// TIA Portal V20 export
DATA_BLOCK "DataFromStandard"   // DB128
// stored: Access Published, InstanceOfName Safety.typeDataToSafety, InstanceOfType UDT, Namespace Safety
"Safety.typeDataToSafety"
   // VAR
   //    ackSafetyFromHmi : Int;
   //    ackSafetyGlobal : Bool;
   //    ackFromUnit1 : Bool;
   //    ackSafetyFromMobileHMI : Bool;
   //    resetSafetyFromMobileHMI : Bool;
   //    connectionBoxID_1 : Int;
   //    connectionBoxID_2 : Int;
   //    MobilePanelConnected : Bool;
   //    MobilePannelPermissions : Bool;
   //    "PhmiNo1.Connected" : Bool;
   //    "PhmiNo2.Connected" : Bool;
   //    KeyBoxStatus : Int;
   //    DeselectBA30 : Bool;
   //    DeselectBA40 : Bool;
   //    DeselectBA15 : Bool;
   //    DeselectBA60 : Bool;
   //    PowerOnCommand : Bool;
   //    leftUnwinderRadius : Int;
   //    rightUnwinderRadius : Int;
   //    PhmiCommunicationOK : Bool;
   //    allBrakeTesting : "Safety.typeBrakeTest";
   //    Unwinder_Left_DiaData : "Safety.typeSafetyDia";
   //    Unwinder_Right_DiaData : "Safety.typeSafetyDia";
   //    FrameCoverSensor : "Safety.SensorStatus";
   //    unitMode : "Safety.typeUnitMode";
   //    unitState : "Safety.typeUnitStatus";
   //    winderUsed : "Safety.typeWinderUseMode";
   //    GateCutter : "Safety.typeFdoorCommands";
   //    GateMagazine : "Safety.typeFdoorCommands";
   //    GateConveyor : "Safety.typeFdoorCommands";
   //    GateCentralAisle : "Safety.typeFdoorCommands";
   //    scrapBox1Interface : "Safety.typeScrapBoxMonitoring";
   //    OpLampStatus : "Safety.typeOpLampStatus";
   //    clock : "Safety.typeGlobalClockMem";
   // END_VAR
BEGIN
END_DATA_BLOCK
